// SIMATIC S7-200 SMART project (STEP 7-Micro/WIN SMART), CPU SR40

SYMBOL_TABLE 系统符号
First_Scan_On    SM0.1    // 仅在第一个扫描周期时接通
END_SYMBOL_TABLE

ORGANIZATION_BLOCK MAIN:OB1
TITLE=程序注释
BEGIN
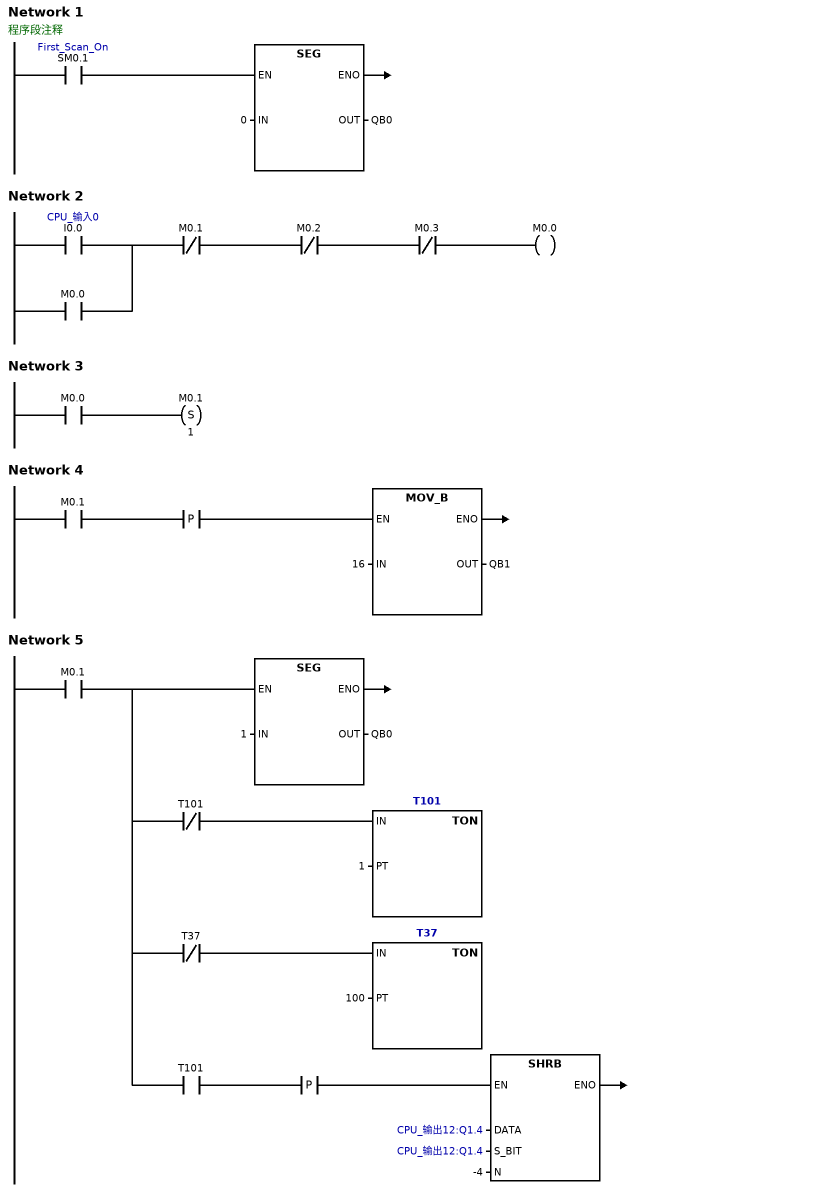
Network 1
// 程序段注释
LD     First_Scan_On:SM0.1
SEG    0, QB0
Network 2
LD     CPU_输入0:I0.0
O      M0.0
AN     M0.1
AN     M0.2
AN     M0.3
=      M0.0
Network 3
LD     M0.0
S      M0.1, 1
Network 4
LD     M0.1
EU
MOVB   16, QB1
Network 5
LD     M0.1
LPS
SEG    1, QB0
AN     T101
TON    T101, 1
LRD
AN     T37
TON    T37, 100
LPP
A      T101
EU
SHRB   CPU_输出12:Q1.4, CPU_输出12:Q1.4, -4
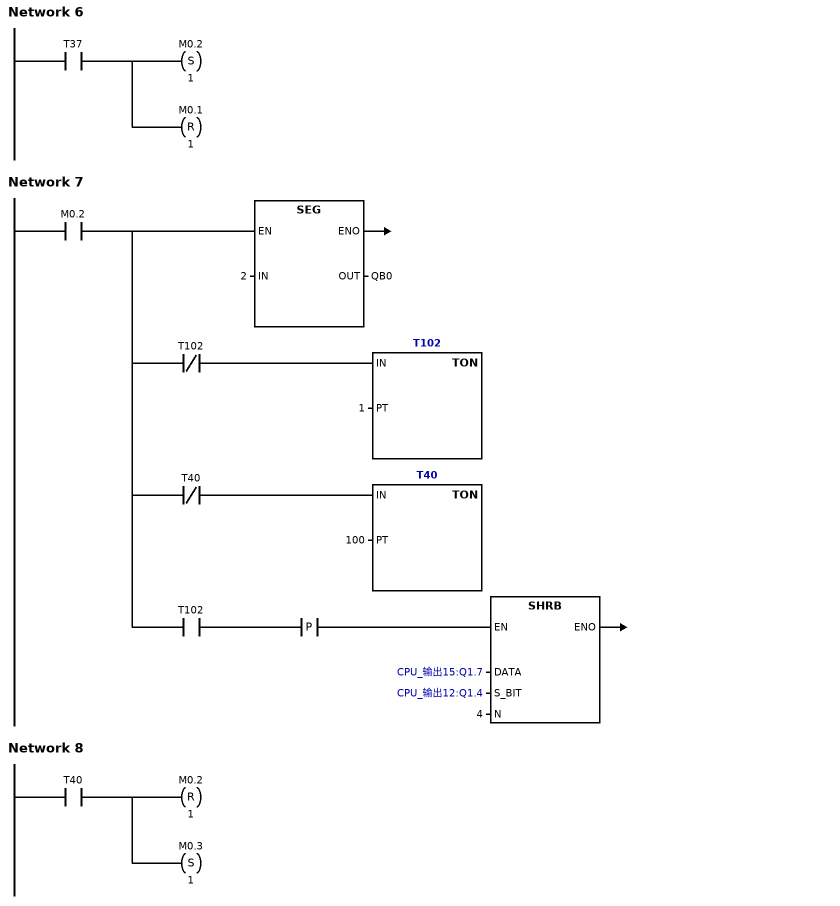
Network 6
LD     T37
S      M0.2, 1
R      M0.1, 1
Network 7
LD     M0.2
LPS
SEG    2, QB0
AN     T102
TON    T102, 1
LRD
AN     T40
TON    T40, 100
LPP
A      T102
EU
SHRB   CPU_输出15:Q1.7, CPU_输出12:Q1.4, 4
Network 8
LD     T40
R      M0.2, 1
S      M0.3, 1
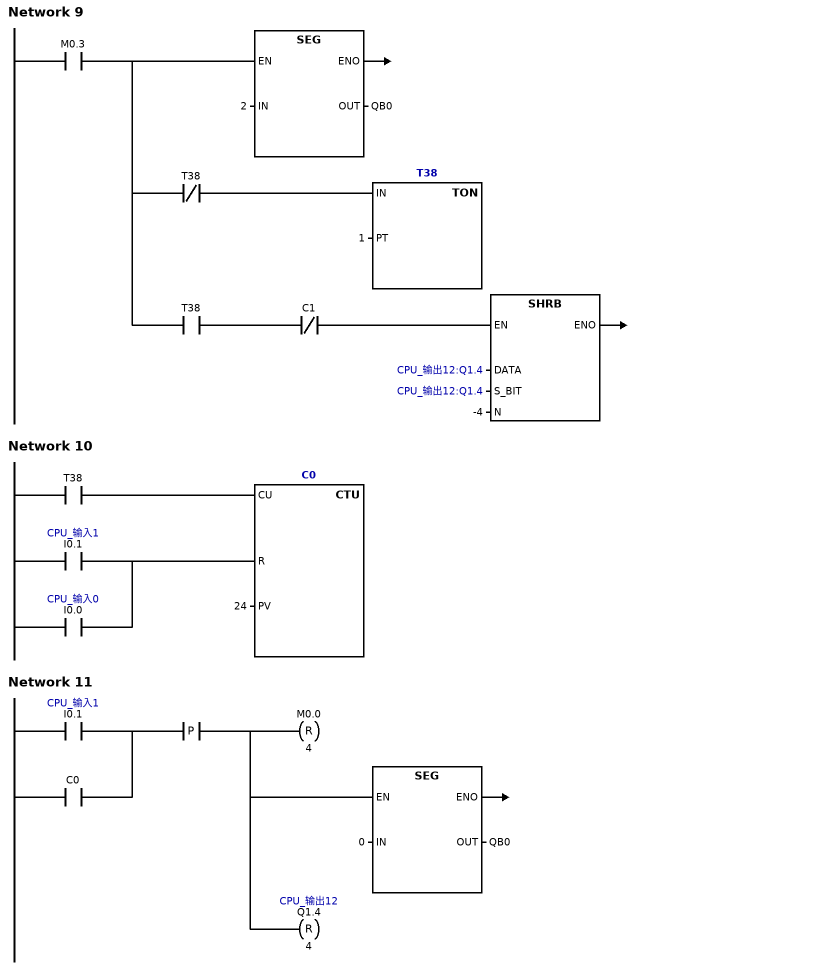
Network 9
LD     M0.3
LPS
SEG    2, QB0
AN     T38
TON    T38, 1
LPP
A      T38
AN     C1
SHRB   CPU_输出12:Q1.4, CPU_输出12:Q1.4, -4
Network 10
LD     T38
LD     CPU_输入1:I0.1
O      CPU_输入0:I0.0
CTU    C0, 24
Network 11
LD     CPU_输入1:I0.1
O      C0
EU
R      M0.0, 4
SEG    0, QB0
R      CPU_输出12:Q1.4, 4
END_ORGANIZATION_BLOCK
